FUNCTION_BLOCK Watchdog
VAR_INPUT
	enable : BOOL;
	
	toggleBit : BOOL;
	timeoutWidth : TIME := DEFAULT_ADS_TIMEOUT;
END_VAR
VAR_OUTPUT
	timeout : BOOL;
END_VAR
VAR	
	timer : TON;
	timerTrig : R_TRIG;
END_VAR

timerTrig(
	CLK:= timerTrig.CLK XOR toggleBit,
	Q=> ); //reset timer

timer(IN:= NOT timerTrig.Q, PT:= timeoutWidth, Q=> timeout, ET=> );

END_FUNCTION_BLOCK

(* stored: Version 1.1.0.1, ProductVersion 3.1.4024.11
   POU Watchdog: Id {5441069f-d199-4420-9a7a-e035c7bf04a5}, SpecialFunc None *)
